TYPE ST_Auto_LowerFeedInConveyorCommand EXTENDS ST_CommandBasic :
STRUCT
END_STRUCT
END_TYPE

(* stored: Version 1.1.0.1, ProductVersion 3.1.4024.13
   DUT ST_Auto_LowerFeedInConveyorCommand: Id {2e635254-e26c-4b49-bdac-bcfa59252132} *)
